TYPE ST_Issue94 :
STRUCT
	BoolValue 	: bool := TRUE;
	ArrayValue 	:  ARRAY [0..1] OF ST_Issue94_Byte := [(ByteValue := 1), (ByteValue := 2)];
END_STRUCT
END_TYPE

(* stored: Version 1.1.0.1, ProductVersion 3.1.4024.12
   DUT ST_Issue94: Id {1998953c-3ab4-49af-990f-42871545692c} *)
